{attribute 'linkalways'} 
{attribute 'no_explicit_call' := 'This FB is a CLASS and must be accessed using methods or properties'}
{attribute 'enable_dynamic_creation'}
FUNCTION_BLOCK Node_F_VN_KeyPointsAndDescriptorsAKAZE EXTENDS VisionNode
VAR
    ipSrcImage : _ITcVnImage;
    ipKeyPoints : _ITcVnContainer;
    ipDescriptors : _ITcVnImage;
    hrPrev : _HRESULT(S_OK);
	hresult : _HRESULT(S_OK);
END_VAR

METHOD PUBLIC  Clone : I_Node
VAR
	pNode : POINTER TO Node_F_VN_KeyPointsAndDescriptorsAKAZE;
END_VAR
pNode := __NEW(Node_F_VN_KeyPointsAndDescriptorsAKAZE);
Clone := pNode^;
END_METHOD

METHOD FB_init : BOOL
VAR_INPUT
	bInitRetains : BOOL; // if TRUE, the retain variables are initialized (warm start / cold start)
	bInCopyCode : BOOL;  // if TRUE, the instance afterwards gets moved into the copy code (online change)
END_VAR
AddInput('ipSrcImage', ipSrcImage);
AddInput('hrPrev', hrPrev);
AddOutput('ipKeyPoints', ipKeyPoints);
AddOutput('ipDescriptors', ipDescriptors);
AddOutput('hresult',hresult);
END_METHOD

METHOD PROTECTED OnExecute
hresult.Value := F_VN_KeyPointsAndDescriptorsAKAZE(
	ipSrcImage := ipSrcImage.Value,
    ipKeyPoints := ipKeyPoints.Value,
    ipDescriptors := ipDescriptors.Value,
	hrPrev:= hrPrev.Value);
END_METHOD

METHOD PUBLIC PreExecutionCheck
VAR_INPUT
	Check : I_PreExecutionChecks;
END_VAR
Check.IsTrue(ipSrcImage.IsValid, 'ipSrcImage must contain an image');
Check.IsTrue(ipSrcImage.HasChannelCount(1), 'ipSrcImage must have 1 channel');
END_METHOD

END_FUNCTION_BLOCK

(* stored: Version 1.1.0.1, ProductVersion 3.1.4024.15
   POU Node_F_VN_KeyPointsAndDescriptorsAKAZE: Id {098e9fad-16d9-04de-0b4d-df10c577e0ad}, SpecialFunc None
   Folder Constructor: Id {70f72208-927e-0ce8-1c01-bea45b00ca70}
   Method Clone: Id {c24f529c-65da-0111-1e03-2293290a3184}
   Method FB_init: Id {0ef9648f-4421-0d75-3e5f-1b1150561826}
   Method OnExecute: Id {d1c30d66-e6da-08a9-15aa-935fd194105d}
   Method PreExecutionCheck: Id {4f46d6d3-a28a-09f8-3e72-b84ed80a4536} *)
